(* IEC 61131-3 sources: Livny/public/Livny, 5 files *)

(* ---- 01_DUT_Types.st ---- *)
(* =========================================================================
   ПРОЕКТ    : Весовой дозатор сахара в мешки 25/50 кг («Ливны»)
   ПЛАТФОРМА : ОВЕН СПК107 · CODESYS 3.5.17 · IEC 61131-3 (Structured Text)
   ОБОРУДОВАНИЕ:
     - МВ110-224.1ТД  — модуль ввода сигнала тензодатчика (вес), RS-485
     - МВ110-8Д.4Р    — 8 дискретных входов / 4 релейных выхода, RS-485
   =========================================================================
   ФАЙЛ      : 01_DUT_Types.st
   НАЗНАЧЕНИЕ: Глобальные типы данных (DUT) проекта.
               В CODESYS: "Добавить объект → DUT", язык ST, перенести типы.
   ========================================================================= *)

TYPE E_DoserState :
(* ------------------------------------------------------------------
   Автомат состояний дозатора. Значения с запасом (шаг 10) —
   удобно для отладки и визуализации СПК107.
   ------------------------------------------------------------------ *)
(
    ST_STOP        := 0,     (* ОСТАНОВ: все выходы отключены            *)
    ST_READY       := 10,    (* ГОТОВНОСТЬ: ожидание команды ПУСК        *)
    ST_CLAMPING    := 20,    (* ЗАЖИМ: фиксация мешка, контроль концевика*)
    ST_TARE        := 30,    (* ТАРА: стабилизация и обнуление веса      *)
    ST_FEED_COARSE := 40,    (* ГРУБО: основная (быстрая) подача сахара  *)
    ST_FEED_FINE   := 50,    (* ТОЧНО: доводка малым питателем           *)
    ST_SETTLING    := 60,    (* УСПОКОЕНИЕ: ожидание стабильного веса    *)
    ST_CHECK       := 70,    (* КОНТРОЛЬ: проверка дозы в допуске        *)
    ST_TOPUP       := 75,    (* ДОСЫПКА: устранение недовеса             *)
    ST_UNCLAMP     := 80,    (* СБРОС: разжим, мешок уходит              *)
    ST_PAUSE       := 90,    (* ПАУЗА: технологическая пауза цикла       *)
    ST_ALARM       := 999    (* АВАРИЯ: требуется вмешательство          *)
);
END_TYPE

TYPE ST_DoseParams :
(* ------------------------------------------------------------------
   Технологические параметры дозирования.
   Загружаются с экрана СПК107 (рецепты 25 / 50 кг), сохраняются
   в RETAIN-области по желанию integratora.
   Все массы — в килограммах (кг), времена — TIME.
   ------------------------------------------------------------------ *)
STRUCT
    rSetpoint       : REAL := 25.0;     (* Заданная масса дозы, кг              *)
    rCoarseCutoff   : REAL := 2.5;      (* Остаток до дозы, на котором
                                           отключается ГРУБАЯ подача, кг
                                           (обычно 8…12 % дозы)                 *)
    rInFlightInit   : REAL := 0.150;    (* Начальная оценка «зависания»
                                           продукта в воздухе/шнеке, кг         *)
    rInFlightMin    : REAL := 0.020;    (* Нижняя граница автокоррекции, кг     *)
    rInFlightMax    : REAL := 0.800;    (* Верхняя граница автокоррекции, кг    *)
    rLearnGain      : REAL := 0.30;     (* Коэффициент обучения 0…1
                                           (доля ошибки, вносимая в коррекцию)  *)
    xLearnEnable    : BOOL := TRUE;     (* Разрешение адаптации «на лету»       *)
    rTolerancePlus  : REAL := 0.050;    (* Допуск «+» на дозу, кг (0,2 % —
                                           жёстче ГОСТ 8.579-2002)              *)
    rToleranceMinus : REAL := 0.050;    (* Допуск «–» на дозу, кг               *)
    rStabBand       : REAL := 0.030;    (* Полоса стабильности весов, кг        *)
    tStabTime       : TIME := T#1S;     (* Время удержания в полосе
                                           стабильности, с                      *)
    tSettle         : TIME := T#1500MS; (* Успокоение после закрытия питателя   *)
    tClampTimeout   : TIME := T#3S;     (* Контроль времени закрытия зажима     *)
    tTareTimeout    : TIME := T#8S;     (* Контроль времени тарирования         *)
    tFlowCheck      : TIME := T#2500MS; (* Окно контроля наличия потока         *)
    rFlowMinStep    : REAL := 0.250;    (* Мин. прирост веса за окно
                                           tFlowCheck на грубой подаче, кг      *)
    rFineFlowMin    : REAL := 0.050;    (* То же для точной подачи, кг          *)
    rTareMax        : REAL := 0.500;    (* Макс. вес пустого мешка (тары), кг   *)
    rTareMin        : REAL := 0.010;    (* Мин. вес пустого мешка (тары), кг    *)
    iTopupMax       : INT  := 3;        (* Макс. число попыток досыпки          *)
    tTopupMax       : TIME := T#2S;     (* Макс. длительность одной досыпки     *)
    tRelease        : TIME := T#800MS;  (* Время разжима (мешок падает)         *)
    tPause          : TIME := T#1S;     (* Пауза перед следующим циклом         *)
    rSetpointMin    : REAL := 5.0;      (* Предел уставки (защита ввода), кг    *)
    rSetpointMax    : REAL := 50.0;     (* Предел уставки (защита ввода), кг    *)
END_STRUCT
END_TYPE

TYPE ST_DoseStats :
(* ------------------------------------------------------------------
   Смена/статистика. Сбрасывается с экрана оператора.
   ------------------------------------------------------------------ *)
STRUCT
    diCount    : DINT := 0;     (* Количество отвешенных доз              *)
    rTotalNet  : REAL := 0.0;   (* Суммарный вес нетто, кг                *)
    rLastNet   : REAL := 0.0;   (* Последняя отвешенная доза, кг          *)
    rLastError : REAL := 0.0;   (* Последняя ошибка (факт − задание), кг  *)
    rSumError  : REAL := 0.0;   (* Сумма ошибок (для среднего), кг        *)
    rMinNet    : REAL := 0.0;   (* Минимальная доза за смену, кг          *)
    rMaxNet    : REAL := 0.0;   (* Максимальная доза за смену, кг         *)
    diUnder    : DINT := 0;     (* Число аварийных недовесов              *)
    diOver     : DINT := 0;     (* Число аварийных передозов              *)
    diTopups   : DINT := 0;     (* Число выполненных досыпок              *)
END_STRUCT
END_TYPE

TYPE ST_Alarms :
(* ------------------------------------------------------------------
   Журнал аварий. Событийные аварии — с самоблокировкой (сброс
   только квитированием), непрерывные условия — «живые».
   ------------------------------------------------------------------ *)
STRUCT
    xEStop      : BOOL;   (* Аварийный останов (грибок/реле безопасности)*)
    xCommLoss   : BOOL;   (* Потеря связи с МВ110-224.1ТД                *)
    xTareFault  : BOOL;   (* Сбой тарирования (нестабильно/тяжёлый мешок)*)
    xNoFlow     : BOOL;   (* Нет потока продукта: затор шнека, пусто     *)
    xOverdose   : BOOL;   (* Передоз сверх допуска (ручная выгрузка)     *)
    xUnderdose  : BOOL;   (* Недовес сверх допуска после досыпок         *)
    xClampFault : BOOL;   (* Зажим не закрылся за отведённое время       *)
    xAirLow     : BOOL;   (* Низкое давление пневмосети («живое»)        *)
    xLevelLow   : BOOL;   (* Нет продукта в расходном бункере («живое»)  *)
    xCoverOpen  : BOOL;   (* Открыта защитная крышка («живое»)           *)
    xActive     : BOOL;   (* Есть хотя бы одна активная авария           *)
END_STRUCT
END_TYPE

TYPE ST_WeightData :
(* ------------------------------------------------------------------
   Обработанные данные весового канала (после FB_WeightChannel).
   ------------------------------------------------------------------ *)
STRUCT
    rNet      : REAL;    (* Вес нетто: фильтр − тара, кг                 *)
    rGross    : REAL;    (* Вес брутто (отфильтрованный), кг             *)
    rTare     : REAL;    (* Текущая тара, кг                             *)
    xStable   : BOOL;    (* Вес стабилен (полоса + время)                *)
    rFlowRate : REAL;    (* Скорость потока продукта, кг/мин             *)
    xCommOK   : BOOL;    (* Связь с тензомодулем в норме                 *)
END_STRUCT
END_TYPE

TYPE ST_ManualMode :
(* ------------------------------------------------------------------
   Ручной режим (пусконаладка): прямое управление выходами с экрана.
   ------------------------------------------------------------------ *)
STRUCT
    xClamp   : BOOL;     (* Зажим мешка                                  *)
    xCoarse  : BOOL;     (* Грубый питатель                              *)
    xFine    : BOOL;     (* Точный питатель                              *)
    xSignal  : BOOL;     (* Сигнальная лампа/зуммер                      *)
    xTare    : BOOL;     (* Тарирование весов                            *)
END_STRUCT
END_TYPE

TYPE ST_HmiDisplay :
(* ------------------------------------------------------------------
   Поля для экрана СПК107 (визуализация). Заполняются в PRG_HMI,
   объекты HMI привязываются к g_Hmi.*
   ------------------------------------------------------------------ *)
STRUCT
    rNet       : REAL;   (* Текущий вес нетто, кг                        *)
    rSetpoint  : REAL;   (* Уставка дозы, кг                             *)
    rLastError : REAL;   (* Ошибка последней дозы, кг                    *)
    rInFlight  : REAL;   (* Текущая автокоррекция «на лету», кг          *)
    rFlowRate  : REAL;   (* Скорость потока, кг/мин                      *)
    diCount    : DINT;   (* Счётчик доз                                  *)
    rLastNet   : REAL;   (* Последняя доза, кг                           *)
    iState     : INT;    (* Номер состояния автомата (для индикации)     *)
    sState     : STRING(16); (* Мнемокод состояния: ГОТОВ, ГРУБО…        *)
    xStable    : BOOL;   (* Индикатор стабильности                       *)
    xCommOK    : BOOL;   (* Индикатор связи с весами                     *)
    xManual    : BOOL;   (* Признак ручного режима                       *)
END_STRUCT
END_TYPE

(* =========================================================================
   КОНЕЦ ФАЙЛА 01_DUT_Types.st
   ========================================================================= *)

(* ---- 02_GVL_Global.st ---- *)
(* =========================================================================
   ПРОЕКТ    : Весовой дозатор сахара в мешки 25/50 кг («Ливны»)
   ПЛАТФОРМА : ОВЕН СПК107 · CODESYS 3.5.17 · IEC 61131-3 (Structured Text)
   =========================================================================
   ФАЙЛ      : 02_GVL_Global.st
   НАЗНАЧЕНИЕ: Глобальный список переменных (GVL).
               В CODESYS: "Добавить объект → Список глобальных переменных",
               язык "GVL в ST", перенести объявления.

   ВАЖНО: переменные НЕ привязаны к физическим входам/выходам (%I/%Q).
          Связка выполняется интегратором в CODESYS:
            g_rWeightRaw    <- выход веса шаблона МВ110-224.1ТД (МХ110)
            g_xDi*          <- дискретные входы шаблона МВ110-8Д.4Р
            g_xDo*          -> релейные выходы шаблона МВ110-8Д.4Р
   ========================================================================= *)

VAR_GLOBAL

    (* ─────────────────────────────────────────────────────────────────
       ВЕСОВОЙ КАНАЛ — МВ110-224.1ТД (адрес в сети RS-485, напр. 16)
       Подключаются к выходам ФБ-шаблона тензомодуля (библиотека
       шаблонов МХ110 / OwenVendorProtocols).
       ───────────────────────────────────────────────────────────────── *)
    g_rWeightRaw     : REAL;      (* Текущий вес от модуля, кг            *)
    g_xWeightValid   : BOOL;      (* Данные достоверны (опрос без ошибок) *)
    g_xWeightErr     : BOOL;      (* Аппаратная ошибка тензомодуля        *)
    g_xTareToModule  : BOOL;      (* Команда «установить ноль» в модуль
                                     (вход Тара/Zero ФБ-шаблона)          *)

    (* ─────────────────────────────────────────────────────────────────
       ДИСКРЕТНЫЕ ВХОДЫ — МВ110-8Д.4Р (адрес в сети RS-485, напр. 17)
       «Сырые» значения каналов DI0…DI7 до антидребезга.
       ───────────────────────────────────────────────────────────────── *)
    g_xDiStart        : BOOL;     (* DI0: кнопка ПУСК (НО, с фиксацией)   *)
    g_xDiStop         : BOOL;     (* DI1: кнопка СТОП (НО)                *)
    g_xDiEStop        : BOOL;     (* DI2: аварийный стоп — НЗ-контакт
                                     (обрыв цепи = авария)                *)
    g_xDiBagPresent   : BOOL;     (* DI3: датчик «мешок в зоне загрузки»  *)
    g_xDiClampClosed  : BOOL;     (* DI4: концевик «зажим закрыт»         *)
    g_xDiAirOK        : BOOL;     (* DI5: реле давления пневмосети ≥ 4 бар*)
    g_xDiLevelOK      : BOOL;     (* DI6: уровень сахара в бункере выше
                                     минимума                             *)
    g_xDiCoverClosed  : BOOL;     (* DI7: защитная крышка закрыта         *)

    (* ─────────────────────────────────────────────────────────────────
       ДИСКРЕТНЫЕ ВЫХОДЫ — реле R0…R3 модуля МВ110-8Д.4Р
       ───────────────────────────────────────────────────────────────── *)
    g_xDoClamp   : BOOL;          (* R0: пневмоклапан зажима мешка        *)
    g_xDoCoarse  : BOOL;          (* R1: грубый питатель (основной шнек)  *)
    g_xDoFine    : BOOL;          (* R2: точный питатель (малый шнек)     *)
    g_xDoSignal  : BOOL;          (* R3: сигнальная лампа / зуммер        *)

    (* ─────────────────────────────────────────────────────────────────
       КОМАНДЫ С ЭКРАНА СПК107 (объекты визуализации пишут сюда)
       ───────────────────────────────────────────────────────────────── *)
    g_xHmiStart    : BOOL;        (* Экранная кнопка ПУСК                 *)
    g_xHmiStop     : BOOL;        (* Экранная кнопка СТОП                 *)
    g_xHmiAck      : BOOL;        (* Квитирование аварий                  *)
    g_xHmiResetStat: BOOL;        (* Сброс статистики смены               *)
    g_xHmiTare     : BOOL;        (* Ручное тарирование                   *)
    g_xHmiRecipe25 : BOOL;        (* Быстрый выбор рецепта 25 кг          *)
    g_xHmiRecipe50 : BOOL;        (* Быстрый выбор рецепта 50 кг          *)
    g_rHmiSetpoint : REAL := 25.0;(* Поле ввода уставки с экрана, кг      *)
    g_xManualMode  : BOOL;        (* Переключатель АВТО / РУЧНОЙ          *)
    g_Manual       : ST_ManualMode; (* Кнопки ручного режима              *)

    (* ─────────────────────────────────────────────────────────────────
       ПРОЦЕССНЫЕ ДАННЫЕ (общие для логики, HMI и архива)
       ───────────────────────────────────────────────────────────────── *)
    g_Params : ST_DoseParams;     (* Технологические параметры            *)
    g_Stats  : ST_DoseStats;      (* Статистика смены                     *)
    g_Alarms : ST_Alarms;         (* Состояние аварий                     *)
    g_Weight : ST_WeightData;     (* Обработанный весовой канал           *)
    g_Hmi    : ST_HmiDisplay;     (* Данные для экрана                    *)
    g_eState : E_DoserState := ST_STOP; (* Текущее состояние автомата     *)

END_VAR

(* =========================================================================
   КОНЕЦ ФАЙЛА 02_GVL_Global.st
   ========================================================================= *)

(* ---- 04_FB_WeightChannel.st ---- *)
(* =========================================================================
   ПРОЕКТ    : Весовой дозатор сахара в мешки 25/50 кг («Ливны»)
   ПЛАТФОРМА : ОВЕН СПК107 · CODESYS 3.5.17 · IEC 61131-3 (Structured Text)
   =========================================================================
   ФАЙЛ      : 04_FB_WeightChannel.st
   НАЗНАЧЕНИЕ: Первичная обработка весового сигнала МВ110-224.1ТД:
                 - контроль связи (watchdog достоверности);
                 - экспоненциальный фильтр (подавление вибраций шнека);
                 - контроль стабильности (полоса + выдержка);
                 - тарирование (смещение нуля + импульс в модуль);
                 - оценка скорости потока (кг/мин) для диагностики затора.

               Примечание: модуль МВ110-224.1ТД имеет собственный
               цифровой фильтр (настраивается в Owen Configurator),
               программный фильтр здесь — второй каскад.
   ========================================================================= *)

FUNCTION_BLOCK FB_WeightChannel

VAR_INPUT
    rWeightRaw  : REAL;     (* «сырой» вес от ФБ-шаблона модуля, кг       *)
    xValid      : BOOL;     (* данные достоверны (опрос без ошибок)       *)
    xError      : BOOL;     (* аппаратная ошибка модуля/датчика           *)
    xTareCmd    : BOOL;     (* запрос тарирования (импульс от автомата)   *)
    xTareManual : BOOL;     (* ручное тарирование с экрана                *)
    rStabBand   : REAL;     (* полоса стабильности, кг                    *)
    tStabTime   : TIME;     (* выдержка в полосе стабильности             *)
    rTaskCycle  : REAL := 0.02; (* цикл задачи ПЛК, с (см. конфигурацию
                                   задачи СПК107, обычно 10…20 мс)        *)
END_VAR

VAR_OUTPUT
    rNet       : REAL;      (* вес нетто (фильтр − тара), кг              *)
    rGross     : REAL;      (* вес брутто (фильтр), кг                    *)
    rTare      : REAL;      (* текущая тара, кг                           *)
    xStable    : BOOL;      (* вес стабилен                               *)
    rFlowRate  : REAL;      (* скорость потока, кг/мин                    *)
    xCommOK    : BOOL;      (* связь с весовым модулем в норме            *)
    xTarePulse : BOOL;      (* импульс «установить ноль» в ФБ модуля      *)
    xTared     : BOOL;      (* тара успешно установлена                   *)
END_VAR

VAR
    rFlt       : REAL;      (* выход ЭМА-фильтра                          *)
    rPrev      : REAL;      (* значение нетто в предыдущем скане          *)
    rDiffEma   : REAL;      (* ЭМА приращения за скан                     *)
    rStabRef   : REAL;      (* опорное значение для полосы стабильности   *)
    rTareOfs   : REAL;      (* смещение тары, кг                          *)
    rK         : REAL := 0.25;   (* коэффициент ЭМА (0…1; меньше — глубже)*)
    rKFlow     : REAL := 0.10;   (* сглаживание оценки скорости           *)
    tonComm    : TON;       (* watchdog связи                             *)
    tonStab    : TON;       (* выдержка стабильности                      *)
    rtTare     : R_TRIG;    (* фронт запроса тарирования                  *)
    tpTare     : TP;        (* импульс команды в модуль                   *)
    xInitDone  : BOOL;      (* флаг первого скана                         *)
END_VAR

(* ---------------------------------------------------------------------
   0. Первый скан: инициализируем фильтр текущим значением,
      чтобы не «догонять» его от нуля.
   --------------------------------------------------------------------- *)
IF NOT xInitDone THEN
    rFlt      := rWeightRaw;
    rPrev     := rWeightRaw;
    rStabRef  := rWeightRaw;
    xInitDone := TRUE;
END_IF

(* ---------------------------------------------------------------------
   1. WATCHDOG СВЯЗИ. Если модуль не отвечает или сообщает ошибку
      дольше 3 с — весовым данным доверять нельзя: автомат дозирования
      будет переведён в аварию (см. FB_DoserControl).
   --------------------------------------------------------------------- *)
tonComm(IN := xValid AND NOT xError, PT := T#3S);
xCommOK := tonComm.Q;

(* ---------------------------------------------------------------------
   2. ЭКСПОНЕНЦИАЛЬНЫЙ ФИЛЬТР:  y[k] = y[k-1] + K·(x[k] − y[k-1])
      При K = 0.25 и цикле 20 мс постоянная времени ≈ 60 мс:
      вибрации от шнека гасятся, фронт насыпки почти не запаздывает.
   --------------------------------------------------------------------- *)
IF xCommOK THEN
    rFlt := rFlt + rK * (rWeightRaw - rFlt);
END_IF

rGross := rFlt;
rNet   := rFlt - rTareOfs;

(* ---------------------------------------------------------------------
   3. СКОРОСТЬ ПОТОКА (кг/мин).
      Приращение за скан усредняется и пересчитывается в минуту.
      Используется автоматом для ранней диагностики «нет потока».
   --------------------------------------------------------------------- *)
IF xCommOK THEN
    rDiffEma := rDiffEma + rKFlow * ((rNet - rPrev) - rDiffEma);
    rPrev    := rNet;
    IF rTaskCycle > 0.001 THEN
        rFlowRate := 60.0 * rDiffEma / rTaskCycle;
    ELSE
        rFlowRate := 0.0;                 (* защита от деления на 0 *)
    END_IF
ELSE
    rFlowRate := 0.0;
END_IF

(* ---------------------------------------------------------------------
   4. КОНТРОЛЬ СТАБИЛЬНОСТИ. Вес считается стабильным, если
      tStabTime подряд не выходит из полосы ±rStabBand вокруг
      опорного значения. Опора обновляется при каждом «выбеге».
   --------------------------------------------------------------------- *)
IF ABS(rNet - rStabRef) > rStabBand THEN
    rStabRef := rNet;
END_IF;

tonStab(IN := (ABS(rNet - rStabRef) <= rStabBand) AND xCommOK,
        PT := tStabTime);
xStable := tonStab.Q;

(* ---------------------------------------------------------------------
   5. ТАРИРОВАНИЕ. Выполняется только на стабильном весе:
      запоминаем брутто как смещение тары и выдаём импульс
      «установить ноль» в ФБ-шаблон модуля (g_xTareToModule),
      чтобы аппаратный и программный нули совпадали.
   --------------------------------------------------------------------- *)
rtTare(CLK := xTareCmd OR xTareManual);

IF rtTare.Q THEN
    IF xStable AND xCommOK THEN
        rTareOfs := rFlt;            (* программная тара            *)
        xTared   := TRUE;
        tpTare(IN := TRUE, PT := T#500MS);   (* импульс в модуль    *)
    ELSE
        xTared := FALSE;             (* условия не выполнены        *)
    END_IF
ELSE
    tpTare(IN := FALSE);
END_IF;

xTarePulse := tpTare.Q;
rTare      := rTareOfs;

(* При потере связи «замораживаем» признак стабильности —
   дозировать на неверных данных запрещено.                          *)
IF NOT xCommOK THEN
    xStable := FALSE;
END_IF

END_FUNCTION_BLOCK

(* =========================================================================
   КОНЕЦ ФАЙЛА 04_FB_WeightChannel.st
   ========================================================================= *)

(* ---- 06_FB_AlarmManager.st ---- *)
(* =========================================================================
   ПРОЕКТ    : Весовой дозатор сахара в мешки 25/50 кг («Ливны»)
   ПЛАТФОРМА : ОВЕН СПК107 · CODESYS 3.5.17 · IEC 61131-3 (Structured Text)
   =========================================================================
   ФАЙЛ      : 06_FB_AlarmManager.st
   НАЗНАЧЕНИЕ: Централизованная обработка аварий.
               - событийные аварии (затор, передоз, сбой тары…) —
                 с самоблокировкой: сбрасываются только КВИТИРОВАНИЕМ;
               - непрерывные условия (аварийный стоп, связь, воздух,
                 уровень, крышка) — отображаются «вживую»;
               - мигалка 1 Гц для сигнальной лампы.
   ========================================================================= *)

FUNCTION_BLOCK FB_AlarmManager

VAR_INPUT
    (* Живые уровни *)
    xEStop       : BOOL;   (* аварийный стоп (НЗ-цепь разомкнута)        *)
    xCommLoss    : BOOL;   (* нет связи с МВ110-224.1ТД                  *)
    xAirOK       : BOOL;   (* давление пневмосети в норме                *)
    xLevelOK     : BOOL;   (* уровень продукта в норме                   *)
    xCoverClosed : BOOL;   (* защитная крышка закрыта                    *)

    (* Импульсные запросы от FB_DoserControl (защёлкиваются) *)
    xReqTareFault  : BOOL;
    xReqNoFlow     : BOOL;
    xReqOverdose   : BOOL;
    xReqUnderdose  : BOOL;
    xReqClamp      : BOOL;

    (* Квитирование оператором (импульс с экрана/кнопки) *)
    xAckAll      : BOOL;
END_VAR

VAR_OUTPUT
    stA        : ST_Alarms; (* структура для HMI и журнала              *)
    xActiveAny : BOOL;      (* есть активная авария                     *)
    xLampBlink : BOOL;      (* мигающий сигнал 1 Гц при аварии          *)
END_VAR

VAR
    tonBlink : TON;          (* генератор мигания                       *)
END_VAR

(* ---------------------------------------------------------------------
   1. СОБЫТИЙНЫЕ АВАРИИ С САМОБЛОКИРОВКОЙ:
      alarm := request OR (alarm AND NOT ack)
   --------------------------------------------------------------------- *)
stA.xTareFault  := xReqTareFault OR (stA.xTareFault  AND NOT xAckAll);
stA.xNoFlow     := xReqNoFlow    OR (stA.xNoFlow     AND NOT xAckAll);
stA.xOverdose   := xReqOverdose  OR (stA.xOverdose   AND NOT xAckAll);
stA.xUnderdose  := xReqUnderdose OR (stA.xUnderdose  AND NOT xAckAll);
stA.xClampFault := xReqClamp     OR (stA.xClampFault AND NOT xAckAll);

(* ---------------------------------------------------------------------
   2. НЕПРЕРЫВНЫЕ УСЛОВИЯ — индицируются, пока причина не устранена.
   --------------------------------------------------------------------- *)
stA.xEStop    := xEStop;
stA.xCommLoss := xCommLoss;
stA.xAirLow   := NOT xAirOK;
stA.xLevelLow := NOT xLevelOK;
stA.xCoverOpen:= NOT xCoverClosed;

(* ---------------------------------------------------------------------
   3. ОБОБЩЁННЫЙ ПРИЗНАК И МИГАЛКА (1 ГЦ, скважность 2).
   --------------------------------------------------------------------- *)
xActiveAny := stA.xEStop    OR stA.xCommLoss  OR stA.xTareFault
           OR stA.xNoFlow   OR stA.xOverdose  OR stA.xUnderdose
           OR stA.xClampFault OR stA.xAirLow  OR stA.xLevelLow
           OR stA.xCoverOpen;

stA.xActive := xActiveAny;

(* Самоперезапускающийся таймер: Q=0.5с / пауза 0.5с → 1 Гц *)
tonBlink(IN := NOT tonBlink.Q, PT := T#500MS);
xLampBlink := tonBlink.Q AND xActiveAny;

END_FUNCTION_BLOCK

(* =========================================================================
   КОНЕЦ ФАЙЛА 06_FB_AlarmManager.st
   ========================================================================= *)

(* ---- 08_PRG_HMI.st ---- *)
(* =========================================================================
   ПРОЕКТ    : Весовой дозатор сахара в мешки 25/50 кг («Ливны»)
   ПЛАТФОРМА : ОВЕН СПК107 · CODESYS 3.5.17 · IEC 61131-3 (Structured Text)
   =========================================================================
   ФАЙЛ      : 08_PRG_HMI.st
   НАЗНАЧЕНИЕ: Сервисная программа интерфейса оператора (встроенный
               7" экран СПК107): защита полей ввода, быстрые рецепты
               25/50 кг, сброс статистики, подготовка отображаемых
               полей g_Hmi.* и мнемокода состояния.

               Объекты визуализации CODESYS привязываются напрямую
               к переменным GVL (g_Hmi.*, g_xHmi*, g_Manual.*).
   ========================================================================= *)

PROGRAM PRG_HMI

VAR
    rtRecipe25 : R_TRIG;
    rtRecipe50 : R_TRIG;
    rtReset    : R_TRIG;
END_VAR

(* ---------------------------------------------------------------------
   1. ЗАЩИТА ПОЛЯ ВВОДА УСТАВКИ (от случайных/зависших значений экрана)
   --------------------------------------------------------------------- *)
g_rHmiSetpoint := LIMIT(g_Params.rSetpointMin, g_rHmiSetpoint, g_Params.rSetpointMax);

(* Передача уставки в технологические параметры *)
g_Params.rSetpoint := g_rHmiSetpoint;

(* ---------------------------------------------------------------------
   2. БЫСТРЫЕ РЕЦЕПТЫ С ЭКРАНА
   --------------------------------------------------------------------- *)
rtRecipe25(CLK := g_xHmiRecipe25);
IF rtRecipe25.Q THEN
    g_rHmiSetpoint := 25.0;     (* мешок 25 кг *)
END_IF

rtRecipe50(CLK := g_xHmiRecipe50);
IF rtRecipe50.Q THEN
    g_rHmiSetpoint := 50.0;     (* мешок 50 кг *)
END_IF

(* ---------------------------------------------------------------------
   3. СБРОС СТАТИСТИКИ СМЕНЫ
   --------------------------------------------------------------------- *)
rtReset(CLK := g_xHmiResetStat);
IF rtReset.Q THEN
    g_Stats.diCount    := 0;
    g_Stats.rTotalNet  := 0.0;
    g_Stats.rLastNet   := 0.0;
    g_Stats.rLastError := 0.0;
    g_Stats.rSumError  := 0.0;
    g_Stats.rMinNet    := 0.0;
    g_Stats.rMaxNet    := 0.0;
    g_Stats.diUnder    := 0;
    g_Stats.diOver     := 0;
    g_Stats.diTopups   := 0;
END_IF

(* ---------------------------------------------------------------------
   4. ОТОБРАЖАЕМЫЕ ПОЛЯ ЭКРАНА
   --------------------------------------------------------------------- *)
g_Hmi.rNet       := g_Weight.rNet;
g_Hmi.rSetpoint  := g_Params.rSetpoint;
g_Hmi.rLastError := g_Stats.rLastError;
g_Hmi.rFlowRate  := g_Weight.rFlowRate;
g_Hmi.diCount    := g_Stats.diCount;
g_Hmi.rLastNet   := g_Stats.rLastNet;
g_Hmi.iState     := TO_INT(g_eState);
g_Hmi.xStable    := g_Weight.xStable;
g_Hmi.xCommOK    := g_Weight.xCommOK;
g_Hmi.xManual    := g_xManualMode;

(* Мнемокод состояния для строки статуса *)
CASE g_eState OF
    ST_STOP:        g_Hmi.sState := 'СТОП';
    ST_READY:       g_Hmi.sState := 'ГОТОВ';
    ST_CLAMPING:    g_Hmi.sState := 'ЗАЖИМ';
    ST_TARE:        g_Hmi.sState := 'ТАРА';
    ST_FEED_COARSE: g_Hmi.sState := 'ГРУБО';
    ST_FEED_FINE:   g_Hmi.sState := 'ТОЧНО';
    ST_SETTLING:    g_Hmi.sState := 'УСПОК';
    ST_CHECK:       g_Hmi.sState := 'КОНТР';
    ST_TOPUP:       g_Hmi.sState := 'ДОСЫП';
    ST_UNCLAMP:     g_Hmi.sState := 'СБРОС';
    ST_PAUSE:       g_Hmi.sState := 'ПАУЗА';
    ST_ALARM:       g_Hmi.sState := 'АВАРИЯ';
ELSE
    g_Hmi.sState := '---';
END_CASE

END_PROGRAM

(* =========================================================================
   КОНЕЦ ФАЙЛА 08_PRG_HMI.st
   ========================================================================= *)
